{attribute 'qualified_only'}
{attribute 'strict'}
{attribute 'to_string'}
TYPE IOExpantionLocation_t :
( 
	ROOT := 0, // this is the main IO master
	EXPANTION  // this is the expantion of the IO master
);
END_TYPE

(* stored: Version 1.1.0.1
   EnumerationTextList IOExpantionLocation_t: Id {ad364000-4d4e-40eb-b317-1c885842efc5} *)
